// TIA Portal V20 export
VAR_GLOBAL   // PLC tag table "MabsEmptyLine"
   "MABS_J1.6.1_IN" AT %I839.0 : "Global.IB_P01_02_03_in_64bytes_struct";
   "MABS_J1.6.1_Out" AT %Q761.0 : "Global.IB_P01_02_03_out_64bytes_struct";
   "MABS_J1.6.2_IN" AT %I903.0 : "Global.IB_P01_02_03_in_64bytes_struct";
   "MABS_J1.6.2_Out" AT %Q825.0 : "Global.IB_P01_02_03_out_64bytes_struct";
END_VAR
